VISUALIZATION mssgbox  // 200x100
END_VISUALIZATION

(* stored: Version 1.1.0.1, ProductVersion 3.1.4022.12
   Visu mssgbox: Id {8e661b62-a72c-46d3-853c-8242d3aed9f0} *)
